PROGRAM PickAndPlaceUnit
VAR	
	// Rotating table motor M1
    fbRotatingTable: FB_Motor;       	
	bRotatingTableAlarmSignal: BOOL := TRUE;  					  // NC alarm input from the rotating table motor M1
	bRotatingTableRun: BOOL;                  					  // Output to run the the rotating table motor M1  
	bRotatingTableError: BOOL;    			  					  // The rotating table motor M1 is in error state
	
	fbRotationMeasuringTimer: TON;            					  // Timer to measure the time period between the sensor S inputs 
	bMeasureRotation: BOOL;                   					  // Measure the time period between the sensor S inputs for parts 1-3
	tSegmentRotationTime: TIME;               					  // Duration of the rotation to 60 degrees (for one part)
	tTimeToRotateForInit: TIME;									  // Duration of the rotation after the error stop to init the rotating table if we simulate the part sensor signal
	fbInitRotationTimer: TON;									  // Timer for the rotation after the error stop to init the rotating table if we simulate the part sensor signal
	bInitRotationTableByTimer: BOOL;
	
	bUseTimerFeedback: BOOL;	              					  // Use sensor signal simulation if the part counter is greater then a half of parts amount
	fbSegmentRotationTimer: TON;              					  // Sensor signal simulation timer	
	
	// Part sensor S
	fbPartSensor: FB_Sensor;                  
	bPartSensorSignal: BOOL;      			                      // Digital input from sensor S
	
	// Gripper G
	fbGripper: FB_Gripper;        
	bGripperClose: BOOL;          			  					  // Output to close gripper G
	
	// Linear slider motor M2
	fbLinearSlider: FB_LinearMotor;           
	bLinearSliderAlarmSignal: BOOL := TRUE;   					  // NC alarm input from the linear slider motor M2
	bLinearSliderMoveToPick: BOOL;            					  // Output to run the linear slider motor M2  
	bLinearSliderMoveToPlace: BOOL;   	      					  // Output to reverse the linear slider motor M2 
	bLinearSliderError: BOOL;                 					  // The linear slider motor M2 is in error state
	
	// Picking position sensor EP2 of linear slider
	fbLinearSliderPickPosSensor: FB_Sensor;    
	bLinearSliderPickPosSignal: BOOL;         					  // Digital input from sensor EP2     
	
	// Placing position sensor EP1 of linear slider
	fbLinearSliderPlacePosSensor: FB_Sensor;   
	bLinearSliderPlacePosSignal: BOOL;		  					  // Digital input from sensor EP2     
		
	// Process flow
	eStateMachine: eSmPickAndPlace;   							  // State machine for the sequence
	uPartsCounter: UINT := 0;                   				  // Parts counter	
	bStartSequence: BOOL;	                    			      // Start the sequence signal
	fbSensorsSimulation: FB_SensorsSimulation;  				  // Simulate all the sensors signals
	
	Counter :INT := 0;
	FromExchange: INT := 0;
END_VAR

VAR CONSTANT
	SIMULATION_PART_SENSOR_DELAY: TIME:= T#5S;                    // Simulation delay for part sensor S
	SIMULATION_LINEAR_SLIDER_PICK_POS_SENSOR_DELAY: TIME:= T#3S;  // Simulation delay for picking position sensor EP2 of linear slider
	SIMULATION_LINEAR_SLIDER_PLACE_POS_SENSOR_DELAY: TIME:= T#3S; // Simulation delay for placing position sensor EP1 of linear slider
	
	PARTS_AMOUNT: UINT := 6;                                      // Amount of the parts on the table 
END_VAR

{region "Instances call"}
fbRotatingTable(bAlarmSignal := bRotatingTableAlarmSignal,
			  	bRun => bRotatingTableRun, 
		      	bError => bRotatingTableError);
				   
fbRotationMeasuringTimer(IN:= bMeasureRotation, 
						 PT:= T#49D17H2M47S295MS, 
						 Q=> , 
						 ET=> );
							  
fbSegmentRotationTimer(IN:= bUseTimerFeedback, 
					   PT:= tSegmentRotationTime, 
					   Q=> , 
					   ET=> );
							
fbInitRotationTimer(IN:= bInitRotationTableByTimer, 
					PT:= tTimeToRotateForInit, 
					Q=> , 
					ET=> );
	
fbPartSensor(bSignal := bPartSensorSignal, 
			 eSignalType := eSensorType.NO);
			 			 
fbGripper(bClose => bGripperClose);

fbLinearSlider(bAlarmSignal := bLinearSliderAlarmSignal, 
				bMoveToPick => bLinearSliderMoveToPick, 
				bMoveToPlace => bLinearSliderMoveToPlace, 
				bError => bLinearSliderError);
				
fbLinearSliderPickPosSensor(bSignal := bLinearSliderPickPosSignal, 
			 eSignalType := eSensorType.NO);
			 
fbLinearSliderPlacePosSensor(bSignal := bLinearSliderPlacePosSignal, 
			 eSignalType := eSensorType.NO);
			 
{endregion}
			  
{region "Sensors simulation"}


fbSensorsSimulation(bEnable := bStartSequence,
					bRotateTable := bRotatingTableRun,
					bLinearSliderMoveToPick := bLinearSliderMoveToPick,
					bLinearSliderMoveToPlace := bLinearSliderMoveToPlace,
					tPartSensorDelay := SIMULATION_PART_SENSOR_DELAY,
					tLinearSliderPickPosSensorDelay := SIMULATION_LINEAR_SLIDER_PICK_POS_SENSOR_DELAY,
					tLinearSliderPlacePosSensorDelay := SIMULATION_LINEAR_SLIDER_PLACE_POS_SENSOR_DELAY,
					bPartSensorSignal => bPartSensorSignal,
					bLinearSliderPickPosSensorSignal => bLinearSliderPickPosSignal,
					bLinearSliderPlacePosSensorSignal => bLinearSliderPlacePosSignal);
						 
bPartSensorSignal := fbSensorsSimulation.bPartSensorSignal AND NOT (bUseTimerFeedback OR bInitRotationTableByTimer);
						 
{endregion}

{region "State machine"}			  
CASE eStateMachine OF 
	eSmPickAndPlace.STANDSTILL:                                                // SM: All the devices are disabled, waiting for start sequence	
		fbRotatingTable.Stop();                                 
		fbLinearSlider.Stop();
		fbGripper.Open();
		
		IF bStartSequence THEN
			eStateMachine := eSmPickAndPlace.INIT;                             // Activatr INIT state
		END_IF;

		
	eSmPickAndPlace.INIT:									                   // SM: Move the devices to the initial state
		 
		IF fbLinearSliderPlacePosSensor.isFree THEN                            // Move the linear slider to the place position
			fbLinearSlider.MoveToPlace();
		ELSIF fbLinearSliderPlacePosSensor.isOccupied THEN
			fbLinearSlider.Stop();
		END_IF;
				
		IF fbPartSensor.isFree AND fbLinearSliderPlacePosSensor.isOccupied THEN // Rotate the table untill we detect the part
			fbRotatingTable.Run();
			IF tTimeToRotateForInit <> T#0S THEN
				bInitRotationTableByTimer := TRUE;
			END_IF;
		ELSIF fbPartSensor.isOccupied OR fbInitRotationTimer.Q THEN
			fbRotatingTable.Stop();
			tTimeToRotateForInit := T#0S;	 
			bInitRotationTableByTimer := FALSE;		 
						  
			eStateMachine := eSmPickAndPlace.PICK;			                   // Activate PICK state
		END_IF;
			
		IF fbRotatingTable.inError OR fbLinearSlider.inError THEN              // Error handler
			eStateMachine := eSmPickAndPlace.ERROR;                            // Activate ERROE state
		END_IF
		
			 
	eSmPickAndPlace.PICK:	                           						   // SM: picking the part
		IF fbLinearSliderPickPosSensor.isFree THEN
			fbLinearSlider.MoveToPick();                                       // Move the linear slider to the pick position
		ELSIF fbLinearSliderPickPosSensor.isOccupied THEN
			fbLinearSlider.Stop();
			fbGripper.Close();                                                 // Close the gripper at the picking position
			eStateMachine := eSmPickAndPlace.PLACE;	                           // Activate PLACE step
		END_IF;
		
		IF fbLinearSlider.inError THEN										   // Error handler
			eStateMachine :=  eSmPickAndPlace.ERROR;						   // Activate ERROR state
		END_IF;

	 
	eSmPickAndPlace.PLACE:													   // SM: 	
		IF fbLinearSliderPlacePosSensor.isFree THEN								
			fbLinearSlider.MoveToPlace();									   // Move the linear slider to the place position
		ELSIF fbLinearSliderPlacePosSensor.isOccupied THEN
			fbLinearSlider.Stop();
			fbGripper.Open();  												   // Open the gripper
			uPartsCounter := uPartsCounter + 1;								   // Increase the parts counter
			
			IF uPartsCounter < PARTS_AMOUNT THEN											
				eStateMachine := eSmPickAndPlace.ROTATE_TABLE;				   // Activate ROTATE_TABLE step if the parts counter us less than parts amount
			ELSE
				uPartsCounter := 0;
				bStartSequence := FALSE;
				eStateMachine := eSmPickAndPlace.STANDSTILL;                   // Activate STANDSTILL step if all the parts are done
			END_IF;
		END_IF;
		
		IF fbLinearSlider.inError THEN										   // Error handler
			eStateMachine :=  eSmPickAndPlace.ERROR;						   // Activate ERROR state
		END_IF
		
			 
	eSmPickAndPlace.ROTATE_TABLE:                                              // SM: rotate the table
		IF uPartsCounter <= PARTS_AMOUNT/2 THEN			                       // If parts counter is less then half of the part amount then 
			IF fbPartSensor.isFree THEN
				fbRotatingTable.Run();                                         // Rotate the table untill the part sensor signal
				bMeasureRotation := TRUE;                                      // Measure the time between the part sensor signals
			ELSIF fbPartSensor.isOccupied THEN			
				fbRotatingTable.Stop();	
			
				tSegmentRotationTime := fbRotationMeasuringTimer.ET;		   // Store the time between the part sensor signals 
				bMeasureRotation := FALSE;
				
				eStateMachine := eSmPickAndPlace.PICK;			               // Activate PICK step
			END_IF;
		ELSE																   // If parts counter is greater then half of the part amount then
			bUseTimerFeedback := TRUE;                                         // Use the timer to simulate the part sensor signal
			fbRotatingTable.Run();
			IF fbSegmentRotationTimer.Q THEN
				bUseTimerFeedback := FALSE;
				fbRotatingTable.Stop();	
				eStateMachine := eSmPickAndPlace.PICK;                         // Activate PICK step
			END_IF;	
		END_IF; 
		
		IF fbRotatingTable.inError THEN										   // Error handler
				 
			bMeasureRotation := FALSE;		
			IF 	bUseTimerFeedback = TRUE THEN
				tTimeToRotateForInit := tSegmentRotationTime - fbSegmentRotationTimer.ET; 
			END_IF;
			bUseTimerFeedback := FALSE;
			eStateMachine :=  eSmPickAndPlace.ERROR;						   // Activate ERROR state
		END_IF	
		
		
	eSmPickAndPlace.ERROR:													   // SM: unit is in error
		bStartSequence := FALSE;											   // Stop the sequence 
		eStateMachine := eSmPickAndPlace.STANDSTILL;						   // Activate STANDSTILL
END_CASE
{endregion}
	 
	 Counter := Counter + 8;
	 GVL_TcpExchange.uWriteData_PlcTask := Counter;
	 FromExchange := GVL_TcpExchange.uReadData_TcpExchangeTask;

END_PROGRAM

(* stored: Version 1.1.0.1, ProductVersion 3.1.4024.12
   POU PickAndPlaceUnit: Id {74ec56e4-ce97-41cc-a813-656c37416b58}, SpecialFunc None *)
